(* CODESYS project ST2.project

Project tree, tasks and I/O mapping:
  Device : CODESYS Control Win V3, 3S - Smart Software Solutions GmbH, version 3.5.15.30
    application Application
      libraries: Standard, * (System)
      task MainTask (cyclic, interval t#20ms, priority 1) calls PLC_PRG
      task VISU_TASK (cyclic, interval 100 ms, priority 31) calls VisuElems.Visu_Prg
      program PLC_PRG [ST]
      visualisation Visualization
  text list GlobalTextList
*)

// Device/Application/PLC_PRG
PROGRAM PLC_PRG
VAR
	Contact1: BOOL := FALSE;
	Coil1: BOOL := FALSE;
END_VAR

IF Contact1 = TRUE THEN;
	Coil1 := TRUE;
ELSE;
	Coil1 := FALSE;
END_IF;

END_PROGRAM

// Device/Application/Visualization
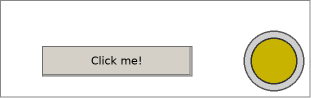
VISUALIZATION Visualization  // 311x98
    Lamp1 (239,26 70x70), variable: PLC_PRG.Coil1, style: Lamp-Lamp1-Yellow
    Button (42,46 150x30), "Click me!"
        tap PLC_PRG.Contact1
END_VISUALIZATION
